PROGRAM AP_V1
VAR
	GetPlate			:Seq_Get_Part;
	SetPlate1			:Seq_Set_Plate_1;
	SetPlate2			:Seq_Set_Plate_2;
	AusrichtenPlates 	:Seq_Ausrichten_Plates;
	SetMountingPlate	:Seq_Set_MPlate;
	AusrichtenMP		:Seq_Ausrichten_MPlate;
END_VAR

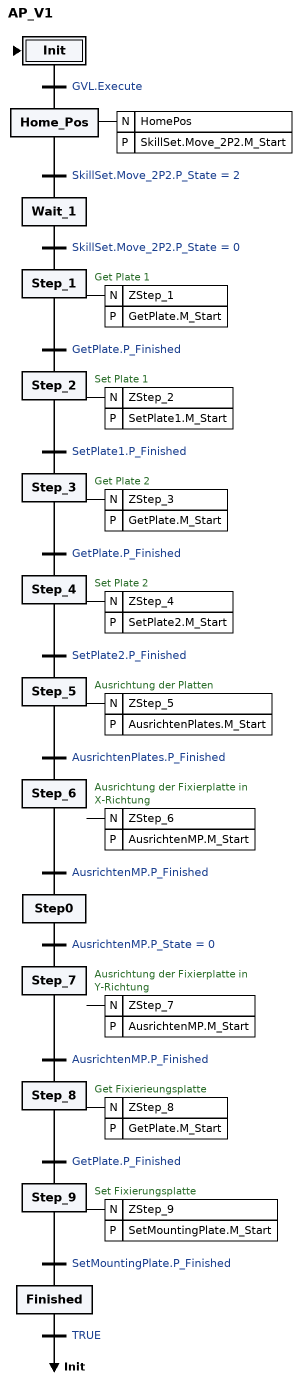
INITIAL_STEP Init:
END_STEP
TRANSITION FROM Init TO Home_Pos
    := GVL.Execute;
END_TRANSITION
STEP Home_Pos:
    HomePos(N);
    SkillSet.Move_2P2.M_Start(P);
END_STEP
TRANSITION FROM Home_Pos TO Wait_1
    := SkillSet.Move_2P2.P_State = 2;
END_TRANSITION
STEP Wait_1:
END_STEP
TRANSITION FROM Wait_1 TO Step_1
    := SkillSet.Move_2P2.P_State = 0;
END_TRANSITION
// Get Plate 1
STEP Step_1:
    ZStep_1(N);
    GetPlate.M_Start(P);
END_STEP
TRANSITION FROM Step_1 TO Step_2
    := GetPlate.P_Finished;
END_TRANSITION
// Set Plate 1
STEP Step_2:
    ZStep_2(N);
    SetPlate1.M_Start(P);
END_STEP
TRANSITION FROM Step_2 TO Step_3
    := SetPlate1.P_Finished;
END_TRANSITION
// Get Plate 2
STEP Step_3:
    ZStep_3(N);
    GetPlate.M_Start(P);
END_STEP
TRANSITION FROM Step_3 TO Step_4
    := GetPlate.P_Finished;
END_TRANSITION
// Set Plate 2
STEP Step_4:
    ZStep_4(N);
    SetPlate2.M_Start(P);
END_STEP
TRANSITION FROM Step_4 TO Step_5
    := SetPlate2.P_Finished;
END_TRANSITION
// Ausrichtung der Platten
STEP Step_5:
    ZStep_5(N);
    AusrichtenPlates.M_Start(P);
END_STEP
TRANSITION FROM Step_5 TO Step_6
    := AusrichtenPlates.P_Finished;
END_TRANSITION
// Ausrichtung der Fixierplatte in X-Richtung
STEP Step_6:
    ZStep_6(N);
    AusrichtenMP.M_Start(P);
END_STEP
TRANSITION FROM Step_6 TO Step0
    := AusrichtenMP.P_Finished;
END_TRANSITION
STEP Step0:
END_STEP
TRANSITION FROM Step0 TO Step_7
    := AusrichtenMP.P_State = 0;
END_TRANSITION
// Ausrichtung der Fixierplatte in Y-Richtung
STEP Step_7:
    ZStep_7(N);
    AusrichtenMP.M_Start(P);
END_STEP
TRANSITION FROM Step_7 TO Step_8
    := AusrichtenMP.P_Finished;
END_TRANSITION
// Get Fixierieungsplatte
STEP Step_8:
    ZStep_8(N);
    GetPlate.M_Start(P);
END_STEP
TRANSITION FROM Step_8 TO Step_9
    := GetPlate.P_Finished;
END_TRANSITION
// Set Fixierungsplatte
STEP Step_9:
    ZStep_9(N);
    SetMountingPlate.M_Start(P);
END_STEP
TRANSITION FROM Step_9 TO Finished
    := SetMountingPlate.P_Finished;
END_TRANSITION
STEP Finished:
END_STEP
TRANSITION FROM Finished TO Init
    := TRUE;
END_TRANSITION

ACTION HomePos:
SkillSet.Move_2P2.P_RobotParam := PunkteZuweisung_Temp.PHome;
END_ACTION

ACTION ZStep_1:
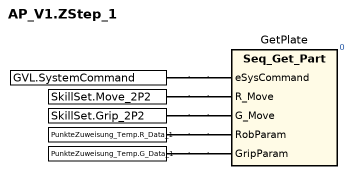
GetPlate(
    eSysCommand := GVL.SystemCommand,
    R_Move := SkillSet.Move_2P2,
    G_Move := SkillSet.Grip_2P2,
    RobParam := PunkteZuweisung_Temp.R_Data_1,
    GripParam := PunkteZuweisung_Temp.G_Data_1); // Seq_Get_Part
END_ACTION

ACTION ZStep_2:
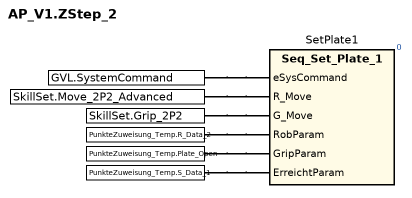
SetPlate1(
    eSysCommand := GVL.SystemCommand,
    R_Move := SkillSet.Move_2P2_Advanced,
    G_Move := SkillSet.Grip_2P2,
    RobParam := PunkteZuweisung_Temp.R_Data_2,
    GripParam := PunkteZuweisung_Temp.Plate_Open,
    ErreichtParam := PunkteZuweisung_Temp.S_Data_1); // Seq_Set_Plate_1
END_ACTION

ACTION ZStep_3:
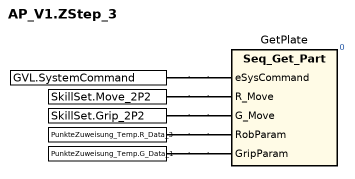
GetPlate(
    eSysCommand := GVL.SystemCommand,
    R_Move := SkillSet.Move_2P2,
    G_Move := SkillSet.Grip_2P2,
    RobParam := PunkteZuweisung_Temp.R_Data_3,
    GripParam := PunkteZuweisung_Temp.G_Data_1); // Seq_Get_Part
END_ACTION

ACTION ZStep_4:
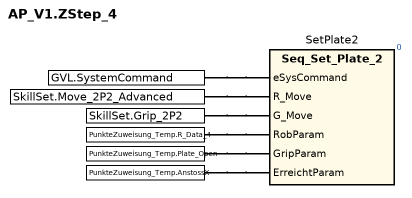
SetPlate2(
    eSysCommand := GVL.SystemCommand,
    R_Move := SkillSet.Move_2P2_Advanced,
    G_Move := SkillSet.Grip_2P2,
    RobParam := PunkteZuweisung_Temp.R_Data_4,
    GripParam := PunkteZuweisung_Temp.Plate_Open,
    ErreichtParam := PunkteZuweisung_Temp.AnstossX); // Seq_Set_Plate_2
END_ACTION

ACTION ZStep_5:
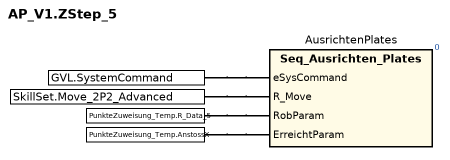
AusrichtenPlates(
    eSysCommand := GVL.SystemCommand,
    R_Move := SkillSet.Move_2P2_Advanced,
    RobParam := PunkteZuweisung_Temp.R_Data_5,
    ErreichtParam := PunkteZuweisung_Temp.AnstossX); // Seq_Ausrichten_Plates
END_ACTION

ACTION ZStep_6:
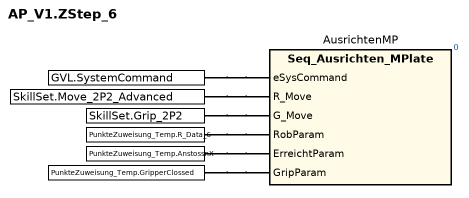
AusrichtenMP(
    eSysCommand := GVL.SystemCommand,
    R_Move := SkillSet.Move_2P2_Advanced,
    G_Move := SkillSet.Grip_2P2,
    RobParam := PunkteZuweisung_Temp.R_Data_6,
    ErreichtParam := PunkteZuweisung_Temp.AnstossnX,
    GripParam := PunkteZuweisung_Temp.GripperClossed); // Seq_Ausrichten_MPlate
END_ACTION

ACTION ZStep_7:
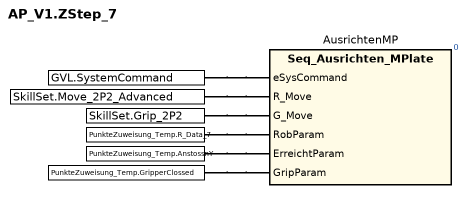
AusrichtenMP(
    eSysCommand := GVL.SystemCommand,
    R_Move := SkillSet.Move_2P2_Advanced,
    G_Move := SkillSet.Grip_2P2,
    RobParam := PunkteZuweisung_Temp.R_Data_7,
    ErreichtParam := PunkteZuweisung_Temp.AnstossnY,
    GripParam := PunkteZuweisung_Temp.GripperClossed); // Seq_Ausrichten_MPlate
END_ACTION

ACTION ZStep_8:
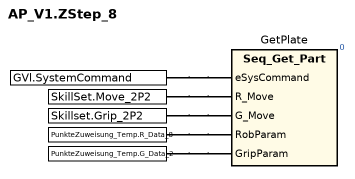
GetPlate(
    eSysCommand := GVl.SystemCommand,
    R_Move := SkillSet.Move_2P2,
    G_Move := Skillset.Grip_2P2,
    RobParam := PunkteZuweisung_Temp.R_Data_8,
    GripParam := PunkteZuweisung_Temp.G_Data_2); // Seq_Get_Part
END_ACTION

ACTION ZStep_9:
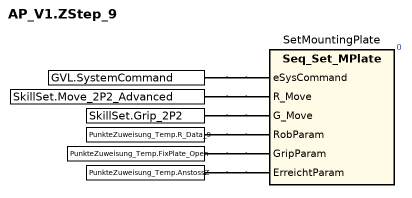
SetMountingPlate(
    eSysCommand := GVL.SystemCommand,
    R_Move := SkillSet.Move_2P2_Advanced,
    G_Move := SkillSet.Grip_2P2,
    RobParam := PunkteZuweisung_Temp.R_Data_9,
    GripParam := PunkteZuweisung_Temp.FixPlate_Open,
    ErreichtParam := PunkteZuweisung_Temp.AnstossZ); // Seq_Set_MPlate
END_ACTION

END_PROGRAM

(* stored: Version 1.1.0.1
   POU AP_V1: Id {3a8a7c03-4d29-456d-873b-3b80c55e380a}, SpecialFunc None
   Folder 01_Zuweisung: Id {ecd5fb79-7da5-47f5-ae11-0167aae7cac7}
   Action HomePos: Id {c0550dcd-88e4-40a1-a94d-79534d55193d}
   Action ZStep_1: Id {4c917d64-6118-40b3-9050-73e978e53fbe}
   Action ZStep_2: Id {79a81c60-47f1-474a-a8cb-80c54df6179e}
   Action ZStep_3: Id {4e88ce0c-50e0-40d7-b6a6-6d376a23ab12}
   Action ZStep_4: Id {97bcf6ff-9d20-4145-9151-e3784d2cb36b}
   Action ZStep_5: Id {3d1f19b9-5918-4f64-8d92-f1d163e92303}
   Action ZStep_6: Id {460557eb-0f9a-4d94-ab8f-3d5181f4a1d4}
   Action ZStep_7: Id {c988377f-7f10-43c2-aec8-be1a575bc717}
   Action ZStep_8: Id {7ca85ed3-2ed0-43f3-a509-74590f78dac8}
   Action ZStep_9: Id {ec4200e9-dac4-4ac0-b77a-54e92ffaa751} *)
